TYPE ST_L7NHA_VelocityCommands :
STRUCT
	VelocitySetpoint	: DINT;	// Target velocity in UU/s used in Profile Velocity mode
END_STRUCT
END_TYPE

(* stored: Version 1.1.0.1, ProductVersion 3.1.4024.15
   DUT ST_L7NHA_VelocityCommands: Id {02a6bae3-040d-47f6-820c-2b500efa1a8c} *)
